// TIA Portal V17 export
// export: Created 2024-09-02T12:50:25.7154996Z, ExportSetting WithDefaults, DisplayName Totally Integrated Automation Portal, DisplayVersion V17, DisplayName TIA Portal Openness, DisplayVersion V17, DisplayName TIA Portal Version Control Interface, DisplayVersion V17, DisplayName STEP 7 Professional, DisplayVersion V17, DisplayName STEP 7 Safety, DisplayVersion V17, DisplayName WinCC Professional, DisplayVersion V17
VAR_GLOBAL   // PLC tag table "CVI3"
   ScrewDriver_IN AT %Q5000.0 : "Desoutter_Input";
   ScrewDriver_OUT AT %I5000.0 : "Desoutter_Output";
END_VAR
